// TIA Portal V20 export
DATA_BLOCK "DB_HMIStatus"   // DB95
{ S7_Optimized_Access := 'TRUE' }
// stored: MemoryReserve 100
   VAR
      WarmUpOn : Bool := FALSE;
      WarmUpTime : Real := 30.0;
      KeyLaserOn : Bool := TRUE;
      Shutter_laser_closed : Bool := FALSE;
      Sonplas : Struct
         LastMeasure : Real;
         CurrentCorrection : Real;
         CouplerOk : Bool;
         Ready : Bool;
      END_STRUCT;
   END_VAR
BEGIN
END_DATA_BLOCK
